FUNCTION_BLOCK BoolArg IMPLEMENTS I_MutBool
VAR
	_val			: BOOL;
END_VAR

PROPERTY Val : BOOL
GET
Val := _val;
END_GET
SET
_val := Val;
END_SET
END_PROPERTY

END_FUNCTION_BLOCK

(* stored: Version 1.1.0.1
   POU BoolArg: Id {e27e2f24-10ad-4112-bcdb-e1d34b1a5e15}, SpecialFunc None
   Property Val: Id {d9f2d2c0-a054-437f-8e42-b9057cb96059}
   Get Get: Id {d4d0bc75-0aba-4584-82fe-08f5e787da5e}
   Set Set: Id {f9b46fd3-d346-4048-a898-ec0e903786b6} *)
